FUNCTION_BLOCK FB_Unit IMPLEMENTS I_Unit
VAR
	Inactive : BOOL;
	iPreviousUnit : I_PreviousUnit;
	iNextUnit : I_NextUnit;
	ForwardDirection : BOOL;
	OldDirection : BOOL;
	
	LED : ARRAY[0..4] OF BOOL;
	
	refCommand : REFERENCE TO E_Command;
	refTon : REFERENCE TO TON;
	UnitNumber : BYTE;
	i : INT;
	
	_Sendable : BOOL;
	_SendStart : BOOL;
	_SendComplete : BOOL;
	
	_Receivable : BOOL;
	_ReceiveStart : BOOL;
	_ReceiveComplete : BOOL;
	
//	SendAbleCounter : INT;
//	SendStartCounter : INT;
//	SendCompleteCounter : INT;
//	ReceiveAbleCounter : INT;
//	ReceiveCompleteCounter : INT;
//	ReceiveStartCounter : INT;
	

	bGenerate : BOOL;
END_VAR

IF NOT __ISVALIDREF(THIS^.refCommand) THEN
	RETURN;
END_IF
IF ForwardDirection <> OldDirection  THEN
	ResetStatus();
END_IF
 OldDirection := ForwardDirection;
MEMSET(ADR(LED),0,SIZEOF(LED));

PROPERTY FirstLED : BOOL
GET
IF ForwardDirection THEN
	FirstLED := LED[0];
ELSE
	FirstLED := LED[4];
END_IF
END_GET
END_PROPERTY

METHOD Initalize
VAR_IN_OUT
	Command : E_Command;
END_VAR
VAR_INPUT
	UnitNumber : BYTE;
	iPreviousUnit : I_PreviousUnit;
	iNextUnit : I_NextUnit;
END_VAR
//THIS^.refTon REF= Ton ;
THIS^.refCommand REF= Command ;
THIS^.UnitNumber := UnitNumber;
THIS^.iPreviousUnit := iPreviousUnit;
THIS^.iNextUnit := iNextUnit;
IF iPreviousUnit = 0 AND iNextUnit = 0 THEN
	Inactive := TRUE;
ELSE
	Inactive := FALSE;
END_IF
END_METHOD

//{attribute 'monitoring' := 'call'}
PROPERTY isReceiveable : BOOL
GET
VAR
	i : BYTE;
END_VAR
isReceiveable := TRUE;
FOR i:=0 TO 4 BY 1 DO
	IF LED[i] = TRUE THEN
		isReceiveable := FALSE;
	END_IF 
END_FOR
END_GET
END_PROPERTY

//{attribute 'monitoring' := 'call'}
PROPERTY isReceiveComplete : BOOL
GET
//isReceiveComplete := iPreviousUnit.isSendComplete;

isReceiveComplete := _ReceiveComplete;
END_GET
END_PROPERTY

//{attribute 'monitoring' := 'call'}
PROPERTY isReceiveStart : BOOL
GET
//isReceiveStart := iPreviousUnit.isSendStart AND NOT iPreviousUnit.isSendComplete;

isReceiveStart := _ReceiveStart;
END_GET
END_PROPERTY

//{attribute 'monitoring' := 'call'}
PROPERTY isSendable : BOOL
GET
//isSendable := LED[4] AND NOT _SendingProduct;
isSendable := _Sendable;
END_GET
END_PROPERTY

//{attribute 'monitoring' := 'call'}
PROPERTY isSendComplete : BOOL
GET
//isSendComplete := isReceiveable;
isSendComplete := _SendComplete;
END_GET
END_PROPERTY

//{attribute 'monitoring' := 'call'}
PROPERTY isSendStart : BOOL
GET
//isSendStart := iNextUnit.isReceiveable AND isSendable AND NOT isReceiveable;
isSendStart := _SendStart;
END_GET
END_PROPERTY

PROPERTY isStopped : BOOL
GET
isStopped := (refCommand = E_Command.Stop) AND NOT _SendStart;
END_GET
END_PROPERTY

PROPERTY LastLED : BOOL
GET
IF ForwardDirection THEN
	LastLED := LED[4];
ELSE
	LastLED := LED[0];
END_IF
END_GET
END_PROPERTY

METHOD ResetStatus
VAR_INPUT
END_VAR
_Sendable 		:=FALSE ;
_SendStart 		:= FALSE;
_SendComplete 	:= FALSE;
_Receivable 	:= FALSE;
_ReceiveStart 	:= FALSE;
_ReceiveComplete:= FALSE;
END_METHOD

METHOD TurnOnLED
VAR_INPUT
	Location : INT;
END_VAR
LED[Location] := TRUE;
END_METHOD

METHOD UpdateStatus
VAR_INPUT
END_VAR
VAR_INST
	FTrig : F_TRIG;
	FTrig2 : F_TRIG;
	FTrig3 : F_TRIG;
	FTrig4 : F_TRIG;
	
	RTrig1 : R_Trig;
	RTrig2 : R_Trig;
	RTrig3 : R_Trig;
	RTrig4 : R_Trig;
	RTrig5 : R_Trig;
	RTrig6 : R_Trig;
END_VAR
ForwardDirection S= refCommand = E_Command.Forward;
ForwardDirection R= refCommand = E_Command.Backward;
_Receivable := isReceiveable;

IF iPreviousUnit <> 0 THEN
	_ReceiveStart := iPreviousUnit.isSendStart;
	_ReceiveComplete := iPreviousUnit.isSendComplete;
END_IF

_Sendable := LastLED;
FTrig(CLK := LastLED);
_SendComplete S= FTrig.Q;

IF iNextUnit <> 0 THEN
	_SendStart S= iNextUnit.isReceiveable AND _Sendable AND NOT (refCommand = E_Command.Stop);
	_SendComplete R= iNextUnit.isReceiveComplete AND NOT FTrig.Q;
	_SendStart R= NOT LastLED;   
END_IF
END_METHOD

END_FUNCTION_BLOCK

(* stored: Version 1.1.0.1, ProductVersion 3.1.4024.12
   POU FB_Unit: Id {69683204-5b7b-42cd-b701-e61dc4d40a10}, SpecialFunc None
   Property FirstLED: Id {2acc34b9-d11a-4f6d-baaf-d3eaaf662191}
   Get Get: Id {8e93fc48-e95c-4164-bc1e-6bccd6c51b16}
   Method Initalize: Id {86c290be-4fb0-45cd-a335-5538d682c0c9}
   Property isReceiveable: Id {eba63f2f-5aa1-460d-87df-77606484889e}
   Get Get: Id {80ded34b-51b0-4685-81ec-7ba7347a80d9}
   Property isReceiveComplete: Id {c98a9f3b-d564-4666-9bbe-10816ecc39e7}
   Get Get: Id {c7034aa0-8716-463a-b878-b681e061f044}
   Property isReceiveStart: Id {ce6ac5ca-944f-4ba7-8c1a-4bec8ad0b98f}
   Get Get: Id {94c32505-5a5d-4603-b4d1-623f625f6e28}
   Property isSendable: Id {355c1b08-215d-4adb-8b4f-13ec17280b46}
   Get Get: Id {ef365e16-57c4-4bd7-b8f3-6e5284c90b90}
   Property isSendComplete: Id {07466405-2512-4777-a8b5-8667bb239141}
   Get Get: Id {93297b68-d385-4162-9731-3fa3d5783167}
   Property isSendStart: Id {ce315785-beb8-49d2-8f45-ba9e51d71840}
   Get Get: Id {5698bef5-05e1-4901-ba41-b0214442e938}
   Property isStopped: Id {b6714c15-a2ac-424d-9a49-ff866afb46f8}
   Get Get: Id {202290ca-ba48-4e4f-810f-843e026f94af}
   Property LastLED: Id {04658c74-e6c0-4ee7-9238-2f1d7aafa07d}
   Get Get: Id {8685b14d-5af9-4859-94ac-35f1d62217f9}
   Method ResetStatus: Id {f40995e1-b50e-4cc6-a2d1-0b8c7435cb54}
   Method TurnOnLED: Id {c38672ba-cb50-44e9-9f51-dd3bde0aa68c}
   Method UpdateStatus: Id {72741a9f-bb73-4834-b36a-7be804a80bc2} *)
